{attribute 'qualified_only'}
VAR_GLOBAL
	fCycleTime : REAL := 0.01;
	fRefPosCylinderVelocity : REAL;
	fRefCylinderStroke : REAL;
	iMaxCylinderStroke : INT := 2;
	iMinCylinderStroke : INT := 0;
	fAutoTime : REAL;
	fManualTime : REAL;
END_VAR

(* stored: Version 1.1.0.1, ProductVersion 3.1.4024.10
   GVL parameter: Id {d2da53b2-7cce-4c80-b396-75a91e644774} *)
